PROGRAM General_Control
VAR
	//	Suunnat HMI luota solun edestä
	Front_door_1				:TON;
	Front_door_2				:TON;
	Right_side_Service_near_1	:TON;
	Right_side_Service_near_2	:TON;
	Right_side_service_far_1	:TON;
	Right_side_service_far_2	:TON;
	Left_side_service_1			:TON;
	Left_side_service_2			:TON;
	Tray_hatch_right			:TON;
	Tray_hatch_right_2			:TON;
	Tray_hatch_right_1			:TON;	
	Tray_hatch_left_1			:TON;
	Tray_hatch_left_2			:TON;
	
	RS_0						:RS;
	RS_1						:RS;
	RS_2						:RS;
	RS_3						:RS;
	RS_4						:RS;
	RS_5						:RS;
	
	Door_locking_time		:TIME:=T#5MS;	//	Oven lukituksen viive
	Door_opening_time		:TIME:=T#1000MS;	//	Oven avauksen viive
	
//	Blinker	
	Blinker_timerON			:TON;
	tempOFF     			:BOOL:=TRUE;
	Blinker1_timerOFF 		:TON;
	tempON    				:BOOL;
	BlinkQ					:BOOL;
	TIME_ON					:TIME:=T#1000MS;
	TIME_OFF				:TIME:=T#1000MS;	
	
//	Blinker fast	
	Blinker_timerON_FAST	:TON;
	tempOFF_FAST     		:BOOL:=TRUE;
	Blinker1_timerOFF_FAST 	:TON;
	tempON_FAST    			:BOOL;
	BlinkQ_FAST				:BOOL;
	TIME_ON_FAST			:TIME:=T#500MS;
	TIME_OFF_FAST			:TIME:=T#500MS;
	
	TON_1					:TON;
	TON_2					:TON;
	VAR1					:BOOL := TRUE;
	VAR2					:BOOL;
	TIMER_TIME				:TIME := T#100MS;
	BlinkQ_RESET			:BOOL;
	
	RS_6: RS;
	RS_7: RS;
	RS_8: RS;
	R_TRIG_0: R_TRIG;
	R_TRIG_1: R_TRIG;
	R_TRIG_2: R_TRIG;
	R_TRIG_3: R_TRIG;
	R_TRIG_4: R_TRIG;
	R_TRIG_5: R_TRIG;
END_VAR
VAR // added by the converter: edge detectors and wires of the graphical bodies
    _w1, _w2, _w3, _w4, _w5 : BOOL;
END_VAR

//Oerlikon projektista kopioitu esimerkkisuoritus

//	Solun modet
	GENERAL.AUTO	:=	HMI.MANUAL_Mode_AUTO;
	GENERAL.MANUAL	:=	HMI.MANUAL_Mode_MANUAL;

//	Programs
	Beacons();
	ButtonBoxes();
	DoorLocks();
	ResetSafety();

//	Blinkers
	BLINK();
	FAST_BLINK();

ACTION Beacons:
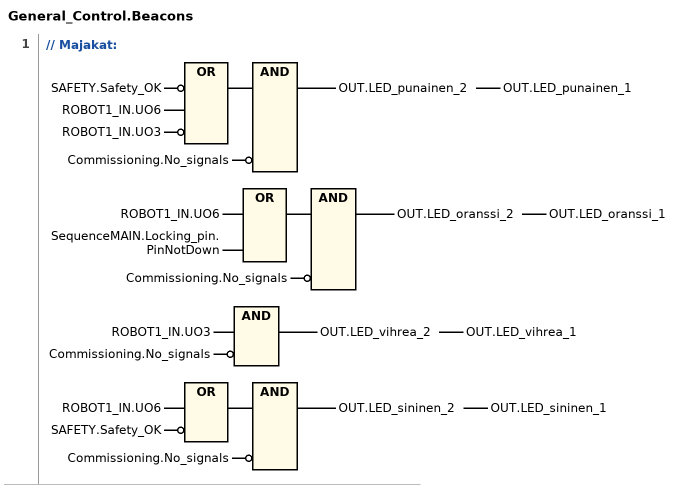
// NETWORK 1
// label: // Majakat
_w1 := (NOT SAFETY.Safety_OK OR ROBOT1_IN.UO6 OR NOT ROBOT1_IN.UO3) AND NOT Commissioning.No_signals;
OUT.LED_punainen_2 := _w1;
OUT.LED_punainen_1 := _w1;
_w2 := (ROBOT1_IN.UO6 OR SequenceMAIN.Locking_pin.PinNotDown) AND NOT Commissioning.No_signals;
OUT.LED_oranssi_2 := _w2;
OUT.LED_oranssi_1 := _w2;
_w3 := ROBOT1_IN.UO3 AND NOT Commissioning.No_signals;
OUT.LED_vihrea_2 := _w3;
OUT.LED_vihrea_1 := _w3;
_w4 := (ROBOT1_IN.UO6 OR NOT SAFETY.Safety_OK) AND NOT Commissioning.No_signals;
OUT.LED_sininen_2 := _w4;
OUT.LED_sininen_1 := _w4;
END_ACTION

ACTION BLINK:
Blinker_timerON(IN:=tempOFF, PT:=TIME_ON);
IF Blinker_timerON.Q THEN
	tempON:=TRUE;
	tempOFF:=FALSE;	
END_IF

Blinker1_timerOFF(IN:=tempON, PT:=TIME_OFF);
IF Blinker1_timerOFF.Q THEN
	tempON:=FALSE;
	tempOFF:=TRUE;
END_IF
BlinkQ :=tempON;
END_ACTION

ACTION ButtonBoxes:
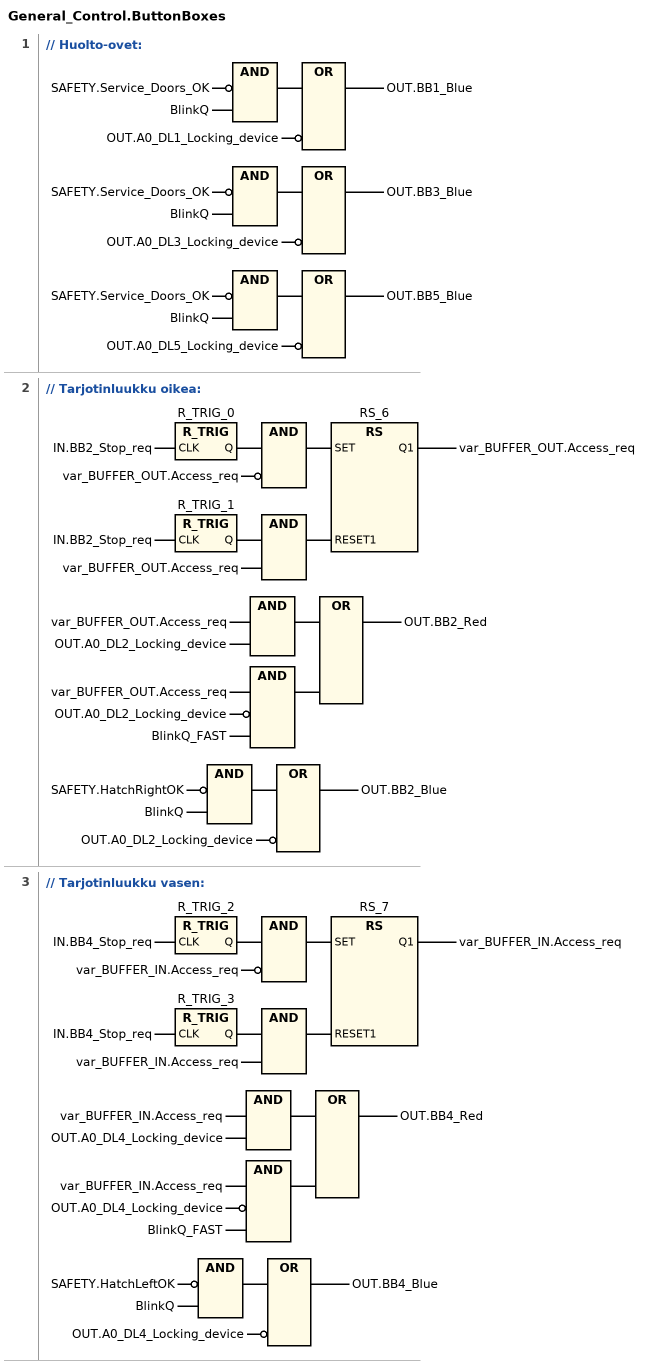
// NETWORK 1
// label: // Huolto-ovet
OUT.BB1_Blue := NOT SAFETY.Service_Doors_OK AND BlinkQ OR NOT OUT.A0_DL1_Locking_device;
OUT.BB3_Blue := NOT SAFETY.Service_Doors_OK AND BlinkQ OR NOT OUT.A0_DL3_Locking_device;
OUT.BB5_Blue := NOT SAFETY.Service_Doors_OK AND BlinkQ OR NOT OUT.A0_DL5_Locking_device;

// NETWORK 2
// label: // Tarjotinluukku oikea
R_TRIG_0(CLK := IN.BB2_Stop_req); // R_TRIG
R_TRIG_1(CLK := IN.BB2_Stop_req); // R_TRIG
RS_6(SET := R_TRIG_0.Q AND NOT var_BUFFER_OUT.Access_req, RESET1 := R_TRIG_1.Q AND var_BUFFER_OUT.Access_req); // RS
var_BUFFER_OUT.Access_req := RS_6.Q1;
OUT.BB2_Red := var_BUFFER_OUT.Access_req AND OUT.A0_DL2_Locking_device OR var_BUFFER_OUT.Access_req AND NOT OUT.A0_DL2_Locking_device AND BlinkQ_FAST;
OUT.BB2_Blue := NOT SAFETY.HatchRightOK AND BlinkQ OR NOT OUT.A0_DL2_Locking_device;

// NETWORK 3
// label: // Tarjotinluukku vasen
R_TRIG_2(CLK := IN.BB4_Stop_req); // R_TRIG
R_TRIG_3(CLK := IN.BB4_Stop_req); // R_TRIG
RS_7(SET := R_TRIG_2.Q AND NOT var_BUFFER_IN.Access_req, RESET1 := R_TRIG_3.Q AND var_BUFFER_IN.Access_req); // RS
var_BUFFER_IN.Access_req := RS_7.Q1;
OUT.BB4_Red := var_BUFFER_IN.Access_req AND OUT.A0_DL4_Locking_device OR var_BUFFER_IN.Access_req AND NOT OUT.A0_DL4_Locking_device AND BlinkQ_FAST;
OUT.BB4_Blue := NOT SAFETY.HatchLeftOK AND BlinkQ OR NOT OUT.A0_DL4_Locking_device;

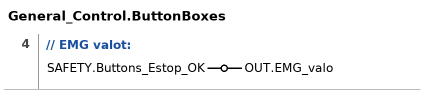
// NETWORK 4
// label: // EMG valot
OUT.EMG_valo := NOT SAFETY.Buttons_Estop_OK;
END_ACTION

ACTION DoorLocks:
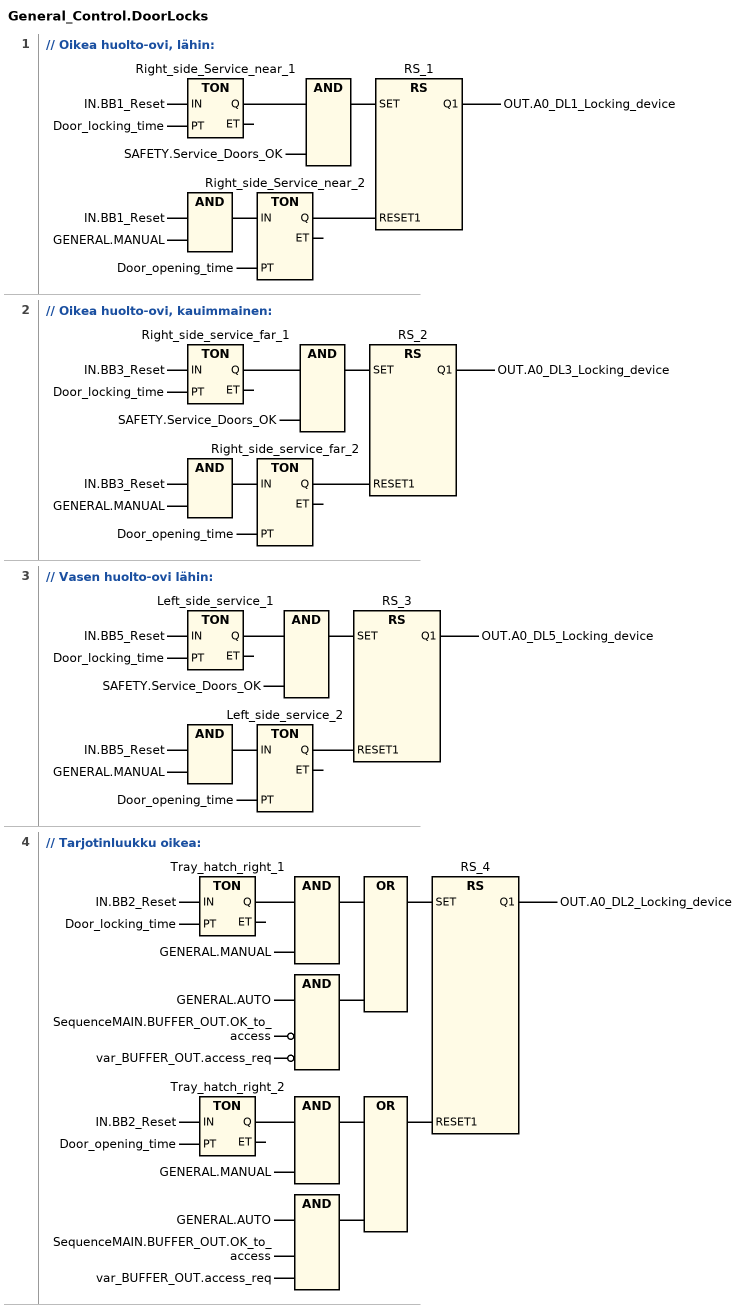
// NETWORK 1
// label: // Oikea huolto-ovi, lähin
Right_side_Service_near_1(IN := IN.BB1_Reset, PT := Door_locking_time); // TON
Right_side_Service_near_2(IN := IN.BB1_Reset AND GENERAL.MANUAL, PT := Door_opening_time); // TON
RS_1(SET := Right_side_Service_near_1.Q AND SAFETY.Service_Doors_OK, RESET1 := Right_side_Service_near_2.Q); // RS
OUT.A0_DL1_Locking_device := RS_1.Q1;

// NETWORK 2
// label: // Oikea huolto-ovi, kauimmainen
Right_side_service_far_1(IN := IN.BB3_Reset, PT := Door_locking_time); // TON
Right_side_service_far_2(IN := IN.BB3_Reset AND GENERAL.MANUAL, PT := Door_opening_time); // TON
RS_2(SET := Right_side_service_far_1.Q AND SAFETY.Service_Doors_OK, RESET1 := Right_side_service_far_2.Q); // RS
OUT.A0_DL3_Locking_device := RS_2.Q1;

// NETWORK 3
// label: // Vasen huolto-ovi lähin
Left_side_service_1(IN := IN.BB5_Reset, PT := Door_locking_time); // TON
Left_side_service_2(IN := IN.BB5_Reset AND GENERAL.MANUAL, PT := Door_opening_time); // TON
RS_3(SET := Left_side_service_1.Q AND SAFETY.Service_Doors_OK, RESET1 := Left_side_service_2.Q); // RS
OUT.A0_DL5_Locking_device := RS_3.Q1;

// NETWORK 4
// label: // Tarjotinluukku oikea
Tray_hatch_right_1(IN := IN.BB2_Reset, PT := Door_locking_time); // TON
Tray_hatch_right_2(IN := IN.BB2_Reset, PT := Door_opening_time); // TON
RS_4(SET := Tray_hatch_right_1.Q AND GENERAL.MANUAL OR GENERAL.AUTO AND NOT SequenceMAIN.BUFFER_OUT.OK_to_access AND NOT var_BUFFER_OUT.access_req, RESET1 := Tray_hatch_right_2.Q AND GENERAL.MANUAL OR GENERAL.AUTO AND SequenceMAIN.BUFFER_OUT.OK_to_access AND var_BUFFER_OUT.access_req); // RS
OUT.A0_DL2_Locking_device := RS_4.Q1;

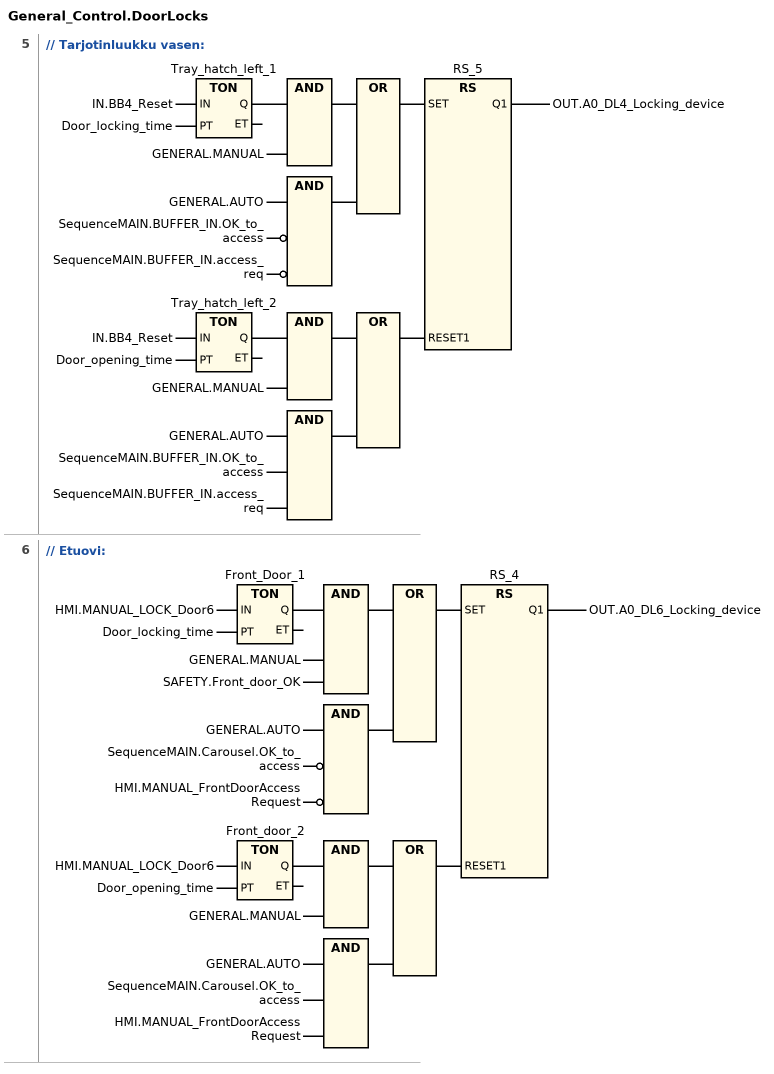
// NETWORK 5
// label: // Tarjotinluukku vasen
Tray_hatch_left_1(IN := IN.BB4_Reset, PT := Door_locking_time); // TON
Tray_hatch_left_2(IN := IN.BB4_Reset, PT := Door_opening_time); // TON
RS_5(SET := Tray_hatch_left_1.Q AND GENERAL.MANUAL OR GENERAL.AUTO AND NOT SequenceMAIN.BUFFER_IN.OK_to_access AND NOT SequenceMAIN.BUFFER_IN.access_req, RESET1 := Tray_hatch_left_2.Q AND GENERAL.MANUAL OR GENERAL.AUTO AND SequenceMAIN.BUFFER_IN.OK_to_access AND SequenceMAIN.BUFFER_IN.access_req); // RS
OUT.A0_DL4_Locking_device := RS_5.Q1;

// NETWORK 6
// label: // Etuovi
Front_Door_1(IN := HMI.MANUAL_LOCK_Door6, PT := Door_locking_time); // TON
Front_door_2(IN := HMI.MANUAL_LOCK_Door6, PT := Door_opening_time); // TON
RS_4(SET := Front_Door_1.Q AND GENERAL.MANUAL AND SAFETY.Front_door_OK OR GENERAL.AUTO AND NOT SequenceMAIN.Carousel.OK_to_access AND NOT HMI.MANUAL_FrontDoorAccessRequest, RESET1 := Front_door_2.Q AND GENERAL.MANUAL OR GENERAL.AUTO AND SequenceMAIN.Carousel.OK_to_access AND HMI.MANUAL_FrontDoorAccessRequest); // RS
OUT.A0_DL6_Locking_device := RS_4.Q1;
END_ACTION

ACTION FAST_BLINK:
Blinker_timerON_FAST(IN:=tempOFF_FAST, PT:=TIME_ON_FAST);
IF Blinker_timerON_FAST.Q THEN
	tempON_FAST:=TRUE;
	tempOFF_FAST:=FALSE;	
END_IF

Blinker1_timerOFF_FAST(IN:=tempON_FAST, PT:=TIME_OFF_FAST);
IF Blinker1_timerOFF_FAST.Q THEN
	tempON_FAST:=FALSE;
	tempOFF_FAST:=TRUE;
END_IF
BlinkQ_FAST :=tempON_FAST;
END_ACTION

ACTION ResetSafety:
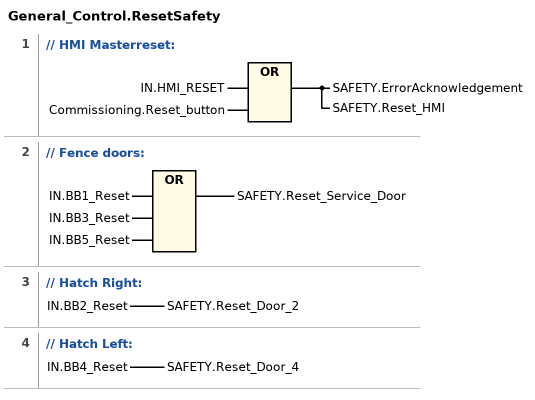
// NETWORK 1
// label: // HMI Masterreset
_w5 := IN.HMI_RESET OR Commissioning.Reset_button;
SAFETY.ErrorAcknowledgement := _w5;
SAFETY.Reset_HMI := _w5;

// NETWORK 2
// label: // Fence doors
SAFETY.Reset_Service_Door := IN.BB1_Reset OR IN.BB3_Reset OR IN.BB5_Reset;

// NETWORK 3
// label: // Hatch Right
SAFETY.Reset_Door_2 := IN.BB2_Reset;

// NETWORK 4
// label: // Hatch Left
SAFETY.Reset_Door_4 := IN.BB4_Reset;
END_ACTION

END_PROGRAM

(* stored: Version 1.1.0.1, ProductVersion 3.1.4024.10
   POU General_Control: Id {65704785-00f0-4323-aba8-d94a6ec4dbe4}, SpecialFunc None
   Folder Blinkers: Id {d3e7d970-ac8d-4ff6-8d7f-b42cbcbe2cf2}
   Action Beacons: Id {5444b389-1f64-45ab-aee0-bbdd68ef2b26}
   Action BLINK: Id {6c05bcf8-7570-4cf8-9373-b1370df401ae}
   Action ButtonBoxes: Id {73f42c4d-85cb-47e5-9a8e-9270ef69d4fb}
   Action DoorLocks: Id {e9598d3f-ab0a-466f-9779-ecebd9c2047e}
   Action FAST_BLINK: Id {180c2814-4b84-4189-93fc-709381e21176}
   Action ResetSafety: Id {0e073681-7ed7-4975-a9b4-28758642255b} *)
